INTERFACE itfSiloFlags

PROPERTY pBufferedWeight : INT
GET
END_GET
SET
END_SET
END_PROPERTY

PROPERTY pLowProduct : BOOL
GET
END_GET
SET
END_SET
END_PROPERTY

PROPERTY pTargetWeight : INT
GET
END_GET
SET
END_SET
END_PROPERTY

END_INTERFACE

(* stored: Version 1.1.0.1, ProductVersion 3.1.4024.12
   Itf itfSiloFlags: Id {f0e8f7a6-5b0c-4c89-a996-d302bb33acab}
   Property pBufferedWeight: Id {1c01fffc-a50b-4524-b76f-77187396020d}
   Get Get: Id {d720b0b4-8384-4260-80aa-e74116bdc981}
   Set Set: Id {caabe211-3b9f-4074-9209-1d88359d61d3}
   Property pLowProduct: Id {e5af26a5-7d76-4e46-b34c-9351d2430ed7}
   Get Get: Id {9cff8734-c7f1-4ab9-83a9-6070a289d53a}
   Set Set: Id {65d36caa-12e0-40f1-a49d-a45852604914}
   Property pTargetWeight: Id {cfdc5047-153d-40cc-b345-266adbe63408}
   Get Get: Id {5304fe68-75b8-4524-8d7f-2e0ee7ebe01d}
   Set Set: Id {7747aad6-5d21-40b6-bbe9-a1fffb871bd1} *)
